// TIA Portal V21 export
VAR_GLOBAL   // PLC tag table "K_ValvoleFesto_VTEM"
END_VAR
VAR_GLOBAL CONSTANT   // user constants
   K_ValvolaFesto_VTEM_LameTaglioCiclo : Int := 1;   // Comando movimento taglio avanti indietro
   K_ValvolaFesto_VTEM_LameTaglioAltezza : Int := 2;   // Comando movimento taglio salita discesa
   K_ValvolaFesto_VTEM_CaricoStecchi : Int := 3;   // Slitta di carico/rifornimento stecchi
   K_ValvolaFesto_VTEM_PreforaturaAghi : Int := 4;   // Comando preforatura con aghi metallici
   K_ValvolaFesto_VTEM_LameTaglioInserimento : Int := 5;   // Comando inserimento lame talgio nel cubo
   K_ValvolaFesto_VTEM_RotazioneStampo : Int := 6;   // Valvola di rotazione cubo avanti e indietro
   K_ValvolaFesto_VTEM_SpintoreStecchi : Int := 7;   // Valvola spintore / inserimento stecchi nel cubo
   "K_ValvolaFesto_VTEM_LameTaglio+Inserimento" : Int := 8;   // Valvola spintore / inserimento stecchi nel cubo
END_VAR
